// TwinCAT 3 PLC project Example
// ProgramVersion: 3.1.4024.12
// libraries:
//   Struckig, * (Stefan Besler)
//   Tc2_Standard, * (Beckhoff Automation GmbH)
//   Tc2_System, * (Beckhoff Automation GmbH)
//   Tc3_Module, * (Beckhoff Automation GmbH)
// project tree:
//   / PlcTask.TcTTO
//   POUs/ Example01_6DoFs.TcPOU, Example02_PositionProfile_2Steps.TcPOU, Example03_2DoFs_Synchronized_Waypoints.TcPOU, Example04_2DoFs_Synchronized_Waypoints_2.TcPOU, Example05_1DoFs_MinDuration.TcPOU, Example06_PhaseSynchronization.TcPOU
// real-time tasks:
//   TASK PlcTask: cycle T#1ms, priority 20, ADS port 350

CONFIGURATION Example
    RESOURCE PLC ON TwinCAT3
        TASK PlcTask(INTERVAL := T#1ms, PRIORITY := 20);
        PROGRAM Example01_6DoFs WITH PlcTask : Example01_6DoFs;
        PROGRAM Example02_PositionProfile_2Steps WITH PlcTask : Example02_PositionProfile_2Steps;
        PROGRAM Example03_2DoFs_Synchronized_Waypoints WITH PlcTask : Example03_2DoFs_Synchronized_Waypoints;
        PROGRAM Example04_2DoFs_Synchronized_Waypoints_2 WITH PlcTask : Example04_2DoFs_Synchronized_Waypoints_2;
        PROGRAM Example05_1DoFs_MinDuration WITH PlcTask : Example05_1DoFs_MinDuration;
        PROGRAM Example06_PhaseSynchronization WITH PlcTask : Example06_PhaseSynchronization;
    END_RESOURCE
END_CONFIGURATION

// ---- POUs/Example01_6DoFs.TcPOU
PROGRAM Example01_6DoFs
VAR
  otg : Struckig.Otg(cycletime:=0.001, dofs:=6) := (
          Synchronization := SynchronizationType.None,
          MaxVelocity :=         [ 1.2,   1.2,  1.2 , 0.6,  0.6, 0.6 ],
          MaxAcceleration :=     [ 4.0,   4.0,  4.0 , 1.5,  1.5, 1.5 ],
          MaxJerk :=             [10.0,  10.0, 10.0,  4.0 , 4.0, 4.0 ],
          CurrentPosition :=     [ 0.0,  -0.1,  0.12, 0.0,  0.3, 0.05],
          CurrentVelocity :=     [ 0.0,   0.0,  0.2,  0.0,  0.0, 0.0 ],
          CurrentAcceleration := [ 0.0,   0.0,  0.0,  0.0,  0.0, 0.0 ],
          TargetPosition :=      [ 1.0,   0.5,  0.5,  0.0, -0.1, 0.2 ],
          TargetVelocity :=      [ 0.0,   0.0,  0.0,  0.0,  0.0, 0.0 ],
          TargetAcceleration :=  [ 0.0,   0.0,  0.0,  0.0,  0.0, 0.0 ]);								
END_VAR

otg(EnableAutoPropagate := TRUE);

END_PROGRAM

// ---- POUs/Example02_PositionProfile_2Steps.TcPOU
PROGRAM Example02_PositionProfile_2Steps
VAR
  otg : Struckig.Otg(cycletime:=0.001, dofs:=1) := (
          Synchronization := SynchronizationType.None,
          MaxVelocity :=         [ 1200.0 ],
          MaxAcceleration :=     [ 25000.0 ],
          MaxJerk :=             [ 25000.0 / 0.008 ],
          CurrentPosition :=     [ 47.0 ],
          CurrentVelocity :=     [ 0.0 ],
          CurrentAcceleration := [ 0.0 ],
          TargetPosition :=      [ 18.0 ],
          TargetVelocity :=      [ -10.0 ],
          TargetAcceleration :=  [ 0.0 ]);                                  
  run : BOOL;
  switched : BOOL;
END_VAR

IF run
THEN  
  // switch to second profile
  otg(EnableAutoPropagate := TRUE);
  IF otg.State = TrajectoryState.Idle AND_THEN NOT switched
  THEN
    switched := TRUE;
    otg.MaxVelocity[0] :=  10.0;
    otg.TargetPosition[0] :=  9.0;
    otg.TargetVelocity[0] :=  0.0;
    otg.TargetAcceleration[0] :=  0.0;
  END_IF
END_IF

END_PROGRAM

// ---- POUs/Example03_2DoFs_Synchronized_Waypoints.TcPOU
PROGRAM Example03_2DoFs_Synchronized_Waypoints
VAR
  otg : Struckig.Otg(cycletime:=0.001, dofs:=2) := (
          Synchronization := SynchronizationType.TimeSync,
          MaxVelocity :=         [ 1000.0, 1000.0 ],
          MaxAcceleration :=     [ 50000.0, 50000.0 ],
          MaxJerk :=             [ 500000.0, 500000.0 ],
          CurrentPosition :=     [ 0.0, 0.0 ],
          CurrentVelocity :=     [ 0.0, 0.0 ],
          CurrentAcceleration := [ 0.0, 0.0 ],
          TargetPosition :=      [ 0.0, 0.0 ],
          TargetVelocity :=      [ 0.0, 0.0 ],
          TargetAcceleration :=  [ 0.0, 0.0 ]);						   
  waypoints : INT := 50;
  a : LREAL := 300;
  b : LREAL := 200;
  w1 : LREAL := 3;
  w2 : LREAL := 2;
  delta : LREAL := PI * 0.5;
  currentWaypoint : INT := 0;
  firstRun : BOOL := TRUE;
  dump : LREAL; // just for testing
END_VAR

// init trajectory
IF firstRun
THEN
  firstRun := FALSE;
  Waypoint(currentWaypoint, px := otg.CurrentPosition[0], py := otg.CurrentPosition[1],
                            vx := otg.CurrentVelocity[0], 
                            vy := otg.CurrentVelocity[1],
                            ax := otg.CurrentAcceleration[0], 
                            ay := otg.CurrentAcceleration[1]
							);

  otg.TargetPosition := otg.CurrentPosition;
  otg.TargetVelocity := otg.CurrentVelocity;
  otg.TargetAcceleration := otg.CurrentAcceleration;  
END_IF

// increment waypoints
otg(EnableAutoPropagate := TRUE);
IF otg.State = TrajectoryState.Idle
THEN
  Waypoint(currentWaypoint, px := otg.TargetPosition[0], py := otg.TargetPosition[1],
                            vx := otg.TargetVelocity[0], 
                            vy := otg.TargetVelocity[1],
                            ax := dump, //otg.Input.TargetAcceleration[0], 
                            ay := dump //otg.Input.TargetAcceleration[1]);
							);
  currentWaypoint := SEL(currentWaypoint + 1 < waypoints, 0, currentWaypoint+1);                    
END_IF

METHOD LissajousCurve
VAR_INPUT
  a : LREAL;
  b : LREAL;
  w1 : LREAL;
  w2 : LREAL;
  delta : LREAL;
  t : LREAL;
END_VAR
VAR_IN_OUT
  px, py : LREAL;
  vx, vy : LREAL;
  ax, ay : LREAL;
END_VAR
px := a * SIN(w1 * t + delta);
py := b * SIN(w2 * t);

vx := a * w1 * COS(w1 * t + delta);
vy := b * w2 * COS(w2 * t);

ax := -a * w1 * w1 * SIN(w1 * t + delta);
ay := -b * w2 * w2 * SIN(w2 * t);
END_METHOD

METHOD Waypoint
VAR_INPUT
  w : INT;
END_VAR
VAR_IN_OUT
  px, py : LREAL;
  vx, vy : LREAL;
  ax, ay : LREAL;
END_VAR
LissajousCurve(a, b, w1, w2, delta, INT_TO_LREAL(w) * 2*PI / INT_TO_LREAL(waypoints),
               px := px, py := py,
               vx := vx, vy := vy,
               ax := ax, ay := ay);
END_METHOD

END_PROGRAM

// ---- POUs/Example04_2DoFs_Synchronized_Waypoints_2.TcPOU
PROGRAM Example04_2DoFs_Synchronized_Waypoints_2
VAR
  otg : Struckig.Otg(cycletime:=0.001, dofs:=2) := (
          Synchronization := SynchronizationType.TimeSync,
          MaxVelocity :=         [ 10.0, 10.0 ],
          MaxAcceleration :=     [ 50000.0, 50000.0 ],
          MaxJerk :=             [ 500000.0, 500000.0 ],
          CurrentPosition :=     [ 0.0, 0.0 ],
          CurrentVelocity :=     [ 0.0, 0.0 ],
          CurrentAcceleration := [ 0.0, 0.0 ],
          TargetPosition :=      [ 0.0, 0.0 ],
          TargetVelocity :=      [ 0.0, 0.0 ],
          TargetAcceleration :=  [ 0.0, 0.0 ]);							   
  waypoints : INT := 50;
  a : LREAL := 300;
  b : LREAL := 200;
  w1 : LREAL := 3;
  w2 : LREAL := 2;
  delta : LREAL := PI * 0.5;
  currentWaypoint : INT := 0;
  firstRun : BOOL := TRUE;
  dump : LREAL; // just for testing
END_VAR

// init trajectory
IF firstRun
THEN
  firstRun := FALSE;
  Waypoint(currentWaypoint, px := otg.CurrentPosition[0], py := otg.CurrentPosition[1],
                            vx := otg.CurrentVelocity[0], 
                            vy := otg.CurrentVelocity[1],
                            ax := otg.CurrentAcceleration[0], 
                            ay := otg.CurrentAcceleration[1]
							);
  otg.TargetPosition := otg.CurrentPosition;
  otg.TargetVelocity := otg.CurrentVelocity;
  otg.TargetAcceleration := otg.CurrentAcceleration;  
END_IF

// increment waypoints
otg(EnableAutoPropagate := TRUE);
IF otg.State = TrajectoryState.Idle
THEN
  Waypoint(currentWaypoint, px := otg.TargetPosition[0], py := otg.TargetPosition[1],
                            vx := otg.TargetVelocity[0], 
                            vy := otg.TargetVelocity[1],
                            ax := dump, //otg.Input.TargetAcceleration[0], 
                            ay := dump //otg.Input.TargetAcceleration[1]);
							);
  currentWaypoint := SEL(currentWaypoint + 1 < waypoints, 0, currentWaypoint+1);
END_IF

METHOD Waypoint
VAR_INPUT
  w : INT;
END_VAR
VAR_IN_OUT
  px, py : LREAL;
  vx, vy : LREAL;
  ax, ay : LREAL;
END_VAR
VAR
  offsetx : LREAL;
END_VAR
offsetx := 10 * TRUNC(ABS(w-1)/2);
w := w MOD 2;
CASE w
OF
  0:
    px := offsetx; py := 0;
    vx := 0; vy := 0;
    ax := 0; ay := 0;
  1:
    px := 100 + offsetx; py := 10;
    vx := 0; vy := 0;
    ax := 0; ay := 0;
END_CASE
END_METHOD

END_PROGRAM

// ---- POUs/Example05_1DoFs_MinDuration.TcPOU
PROGRAM Example05_1DoFs_MinDuration
VAR
  otg : Struckig.Otg(cycletime:=0.001, dofs:=1) := (
          Synchronization := SynchronizationType.TimeSync, // one axis -> no synchronistation is required
          MinDuration := 10.0, // if MinDuration is set to a value > 0 it is considered in trajectory calculation
          MaxVelocity := [ 2000.0 ],
          MaxAcceleration := [ 20000.0 ],
          MaxJerk := [ 800000.0 ],
          CurrentPosition := [ 0 ],
          CurrentVelocity := [ 0 ],
          CurrentAcceleration := [ 0 ],
          TargetPosition := [ 100 ],
          TargetVelocity := [ 0.0, 0.0, 0.0 ],
          TargetAcceleration := [ 0.0, 0.0, 0.0 ]
  );
END_VAR

otg(EnableAutoPropagate := TRUE);

END_PROGRAM

// ---- POUs/Example06_PhaseSynchronization.TcPOU
PROGRAM Example06_PhaseSynchronization
VAR
  otgTimeSync : Struckig.Otg(cycletime:=0.001, dofs:=3) := (
                  Synchronization := SynchronizationType.TimeSync,
                  CurrentPosition :=     [ 0.0, 0.0, 0.0 ],
                  TargetPosition :=      [ 1.0, -1.0, 2.0 ],
                  MaxVelocity :=         [ 1.0, 1.0, 1.0 ],
                  MaxAcceleration :=     [ 1.0, 1.0, 1.0 ],
                  MaxJerk :=             [ 1.0, 1.0, 1.0 ]
  ); 
  
  otgPhaseSync : Struckig.Otg(cycletime:=0.001, dofs:=3) := (
                  Synchronization := SynchronizationType.Phase,
                  CurrentPosition :=     [ 0.0, 0.0, 0.0 ],
                  TargetPosition :=      [ 1.0, -1.0, 2.0 ],
                  MaxVelocity :=         [ 1.0, 1.0, 1.0 ],
                  MaxAcceleration :=     [ 1.0, 1.0, 1.0 ],
                  MaxJerk :=             [ 1.0, 1.0, 1.0 ]
  ); 
  otgTimeSync2 : Struckig.Otg(cycletime:=0.001, dofs:=3) := (
                  Synchronization := SynchronizationType.TimeSync,
                  CurrentPosition :=     [ 0.0, 0.0, 0.0 ],
                  TargetPosition :=      [ 1.0, -1.0, 2.0 ],
                  MaxVelocity :=         [ 1.0, 1.0, 1.0 ],
                  MaxAcceleration :=     [ 1.0, 1.0, 1.0 ]
  ); 
  
  otgPhaseSync2 : Struckig.Otg(cycletime:=0.001, dofs:=3) := (
                  Synchronization := SynchronizationType.Phase,
                  CurrentPosition :=     [ 0.0, 0.0, 0.0 ],
                  TargetPosition :=      [ 1.0, -1.0, 2.0 ],
                  MaxVelocity :=         [ 1.0, 1.0, 1.0 ],
                  MaxAcceleration :=     [ 1.0, 1.0, 1.0 ]
  );   
END_VAR

otgTimeSync(EnableAutoPropagate := TRUE);
otgPhaseSync(EnableAutoPropagate := TRUE);
otgTimeSync2(EnableAutoPropagate := TRUE);
otgPhaseSync2(EnableAutoPropagate := TRUE);

END_PROGRAM
